(* IEC 61131-3 sources: SigmatekTestframework/src/Class/CScreenInterface, 1 file *)

(* ---- CScreenInterface.st ---- *)
(*!
<Class
	Name               = "CScreenInterface"
	Revision           = "0.0"
	RealtimeTask       = "false"
	CyclicTask         = "false"
	BackgroundTask     = "false"
	Sigmatek           = "false"
	OSInterface        = "false"
	HighPriority       = "false"
	Automatic          = "false"
	UpdateMode         = "Prescan"
	SharedCommandTable = "true"
	Objectsize         = "(480,180)">
	<Channels>
		<Server Name="Active" Visualized="false" Initialize="false" WriteProtected="true" Retentive="false"/>
	</Channels>
	<Network Name="CScreenInterface">
		<!-- List of Components in this network -->
		<Components>
			<Object
				Name       = "_base"
				Class      = "_Screen"
				Position   = "(218,120)"
				Visualized = "true"
				Remotely   = "true">
				<Channels>
					<Server Name="Screen"/>
					<Client Name="ImA"/>
					<Client Name="Lse"/>
					<Client Name="No"/>
				</Channels>
			</Object>
		</Components>
		<Comments>
		</Comments>
		<!-- List of Connections in this network -->
		<Connections>
			<Connection Source="this.Screen" Destination="_base.Screen" Vertices="(690,210),(518,210),"/>
			<Connection Source="_base.Lse" Destination="this.Lse" Vertices="(218,210),(30,210),(38,210),"/>
			<Connection Source="_base.No" Destination="this.No" Vertices="(218,270),(38,270),"/>
			<Connection Source="_base.ImA" Destination="this.ImA" Vertices="(218,330),(38,330),"/>
		</Connections>
		<!-- Headerfiles -->
		<Options>
		</Options>
	</Network>
</Class>
*)
#pragma using _Screen

CScreenInterface : CLASS
: _Screen
  //Servers:
	Active 	: SvrCh_DINT;
  //Clients:
  //Variables:
  //Functions:

	FUNCTION VIRTUAL GLOBAL S_End
		VAR_INPUT
			pic 	: ^void;
		END_VAR;

	FUNCTION VIRTUAL GLOBAL S_Start
		VAR_INPUT
			pic 	: ^void;
			firsttime 	: BOOL;
		END_VAR;
  //Tables:
	FUNCTION @STD
		VAR_OUTPUT
			ret_code	: CONFSTATES;
		END_VAR;
	FUNCTION GLOBAL TAB @CT_;
END_CLASS;

//Exclude-SccX
(*
 **********************************************************************
 * \file CScreenInterface.st
 *
 * Interface for Lasal Screen Testing
 * Contains Functions of HMI-Pages
 *
 *
 * Copyright (c) 2016,Hoox.Software, Helmbrechts
 * All Rights Reserved.
 *
 * Created on: 01.06.2016
 *     Author: dressel
 *
 **********************************************************************
 *)

//*****************************************************************************
//
//
//
//
//*****************************************************************************
#pragma warning(disable:73);
FUNCTION VIRTUAL GLOBAL CScreenInterface::S_End
	VAR_INPUT
		pic 	: ^void;
	END_VAR

   Active := 0;

END_FUNCTION

//*****************************************************************************
//
//
//
//
//*****************************************************************************
#pragma warning(disable:73);
FUNCTION VIRTUAL GLOBAL CScreenInterface::S_Start
	VAR_INPUT
		pic 	: ^void;
		firsttime 	: BOOL;
	END_VAR

   Active := 1;

END_FUNCTION
